PROGRAM data_robot_ur3





VAR
	
join_pos_1 : REAL;
join_pos_2 : REAL;
join_pos_3 : REAL;
join_pos_4 : REAL;
join_pos_5 : REAL;
join_pos_6 : REAL;

join_torque_1: REAL;
join_torque_2: REAL;
join_torque_3: REAL;
join_torque_4: REAL;
join_torque_5: REAL;
join_torque_6: REAL;

TCP_pos_x : REAL;
TCP_pos_y : REAL;
TCP_pos_z : REAL;
TCP_pos_rx : REAL;
TCP_pos_ry : REAL;
TCP_pos_rz : REAL;


TCP_force_x : REAL;
TCP_force_y : REAL;
TCP_force_z : REAL;
TCP_torque_x : REAL;
TCP_torque_y : REAL;
TCP_torque_z : REAL;

TCP_force : REAL;

END_VAR





TCP_pos_x := flip_byte(robot_S_ur3.UR_TCP.FLOAT0)*1000;
TCP_pos_y := flip_byte(robot_S_ur3.UR_TCP.FLOAT1)*1000;
TCP_pos_z := flip_byte(robot_S_ur3.UR_TCP.FLOAT2)*1000;
TCP_pos_rx := (flip_byte(robot_S_ur3.UR_TCP.FLOAT3)*180)/PI;
TCP_pos_ry := (flip_byte(robot_S_ur3.UR_TCP.FLOAT4)*180)/PI;
TCP_pos_rz := (flip_byte(robot_S_ur3.UR_TCP.FLOAT5)*180)/PI;


TCP_force  := flip_byte(robot_S_ur3.UR_TCP.FLOAT18);

TCP_force_x := flip_byte(robot_S_ur3.UR_TCP.FLOAT12);
TCP_force_y := flip_byte(robot_S_ur3.UR_TCP.FLOAT13);
TCP_force_z := flip_byte(robot_S_ur3.UR_TCP.FLOAT14);
TCP_torque_x := flip_byte(robot_S_ur3.UR_TCP.FLOAT15);
TCP_torque_y := flip_byte(robot_S_ur3.UR_TCP.FLOAT16);
TCP_torque_z := flip_byte(robot_S_ur3.UR_TCP.FLOAT17);

join_pos_1 := (flip_byte(robot_S_ur3.UR_JOINS.FLOAT0)*180)/PI;
join_pos_2 := (flip_byte(robot_S_ur3.UR_JOINS.FLOAT1)*180)/PI;
join_pos_3 := (flip_byte(robot_S_ur3.UR_JOINS.FLOAT2)*180)/PI;
join_pos_4 := (flip_byte(robot_S_ur3.UR_JOINS.FLOAT3)*180)/PI;
join_pos_5 := (flip_byte(robot_S_ur3.UR_JOINS.FLOAT4)*180)/PI;
join_pos_6 := (flip_byte(robot_S_ur3.UR_JOINS.FLOAT5)*180)/PI;
 
join_torque_1 := flip_byte(robot_S_ur3.UR_float_out.FLOAT0);
join_torque_2 := flip_byte(robot_S_ur3.UR_float_out.FLOAT1);
join_torque_3 := flip_byte(robot_S_ur3.UR_float_out.FLOAT2);
join_torque_4 := flip_byte(robot_S_ur3.UR_float_out.FLOAT3);
join_torque_5 := flip_byte(robot_S_ur3.UR_float_out.FLOAT4);
join_torque_6 := flip_byte(robot_S_ur3.UR_float_out.FLOAT5);

END_PROGRAM

(* stored: Version 1.1.0.1, ProductVersion 3.1.4024.4
   POU data_robot_ur3: Id {6c0eb23f-a835-4ef3-9ad6-2696d3162905}, SpecialFunc None *)
